PROGRAM BB02PL_LineBackground
VAR
END_VAR

MAIN.stLine_BB02PL.fbLine(stLine:=MAIN.stLine_BB02PL);
MAIN.stLine_BB02PL.stStation_BB02PL01.fbStation(
				stLine:=MAIN.stLine_BB02PL,
				stStation:=MAIN.stLine_BB02PL.stStation_BB02PL01);

END_PROGRAM

(* stored: Version 1.1.0.1, ProductVersion 3.1.4024.15
   POU BB02PL_LineBackground: Id {35bf0955-7c31-4039-bfd5-7dc0651238c1}, SpecialFunc None *)
